TYPE UDT_FlowHmi_RD :
STRUCT
  
actStep : UINT; // 当前步号
number : INT; // 流程文本列表编号
name : STRING[20]; // 流程名称
describe : STRING[60]; // 流程说明
  
END_STRUCT
END_TYPE

(* stored: Version 1.1.0.1, ProductVersion 3.1.4024.12
   DUT UDT_FlowHmi_RD: Id {fbe701de-c85b-46de-b9d8-77cfb994e647} *)
